// LS Electric XG5000 project: PLC_1
// PLC LSPLC
// module base 0 slot 0: Input/Output Module:XBC-DR30S (DC 24V Input 18 Contacts, Relay Output 12 Contacts)
// module base 0 slot 9: Analog Input Module:XBO-AD02A (A/D Voltage/Current Input Type(2 Channels))
// module base 0 slot 10: Analog Output Module:XBO-DA02A (D/A Voltage/Current Output Type(2 Channels))

PROGRAM NewProgram (task: Scan Program)

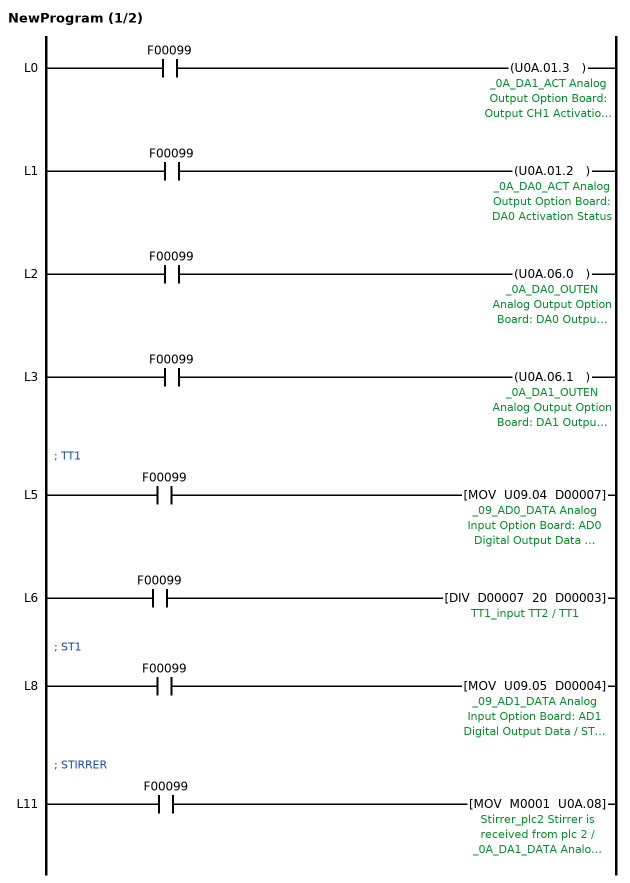
; L0
LOAD      F00099
OUT       U0A.01.3	// _0A_DA1_ACT Analog Output Option Board: Output CH1 Activation Status
; L1
LOAD      F00099
OUT       U0A.01.2	// _0A_DA0_ACT Analog Output Option Board: DA0 Activation Status
; L2
LOAD      F00099
OUT       U0A.06.0	// _0A_DA0_OUTEN Analog Output Option Board: DA0 Output Enable
; L3
LOAD      F00099
OUT       U0A.06.1	// _0A_DA1_OUTEN Analog Output Option Board: DA1 Output Enable
// TT1
; L5
LOAD      F00099
MOV       U09.04 D00007	// _09_AD0_DATA Analog Input Option Board: AD0 Digital Output Data / TT1_input TT2
; L6
LOAD      F00099
DIV       D00007 20 D00003	// TT1_input TT2 / TT1
// ST1
; L8
LOAD      F00099
MOV       U09.05 D00004	// _09_AD1_DATA Analog Input Option Board: AD1 Digital Output Data / ST1 analog input ST1
// STIRRER
; L11
LOAD      F00099
MOV       M0001 U0A.08	// Stirrer_plc2 Stirrer is received from plc 2 / _0A_DA1_DATA Analog Output Option Board: DA1 Digital Input Data

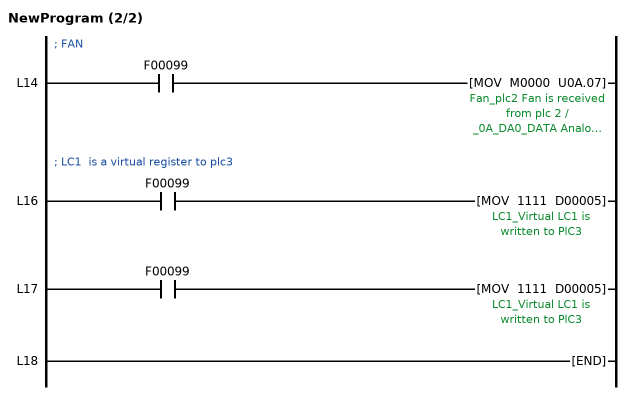
// FAN
; L14
LOAD      F00099
MOV       M0000 U0A.07	// Fan_plc2 Fan is received from plc 2 / _0A_DA0_DATA Analog Output Option Board: DA0 Digital Input Data
// LC1  is a virtual register to plc3
; L16
LOAD      F00099
MOV       1111 D00005	// LC1_Virtual LC1 is written to PlC3 
; L17
LOAD      F00099
MOV       1111 D00005	// LC1_Virtual LC1 is written to PlC3 
; L18
END

VARIABLES AND COMMENTS (devices not used above)
D00002	WORD	fan
K00003	BIT	J1
D00001	WORD	stirrer